{attribute 'GeneratedUsingTerminal: EK1100-0000-0018'}
{attribute addProperty BoxType "EK1100-0000-0018"}
{attribute addProperty Id "Beckhoff_CXxxxxEK1122Beckhoff_CXxxxxEK1122_D04B84CE568"}
{attribute addProperty CRC "2966434434"}
{attribute addProperty Size "568"}
TYPE Beckhoff_CXxxxx_B0D03282 EXTENDS EK1100_AB5A9467 :
STRUCT
	{attribute addProperty Name "Beckhoff_CXxxxxEK1122"}
	{attribute addProperty PreviousPort "Beckhoff CXxxxx : B"}
	Beckhoff_CXxxxxEK1122 : Beckhoff_CXxxxxEK1122_D04B84CE;
END_STRUCT
END_TYPE

(* stored: Version 1.2.0.0, ProductVersion 3.1.4024.9
   DUT Beckhoff_CXxxxx_B0D03282: Id {66a91bed-a658-488f-81ef-38118895b4f7} *)
